// TIA Portal V19 export
FUNCTION "LSW_INTERLOCK" : Void   // FC9, LAD
{ S7_Optimized_Access := 'TRUE' }
// stored: SetENOAutomatically false
   VAR_TEMP   // added for the SCL form of the ladder/FBD networks
      _w1 : Bool;
      _w2 : Bool;
   END_VAR
BEGIN

REGION Network 1: FORWARD LSW
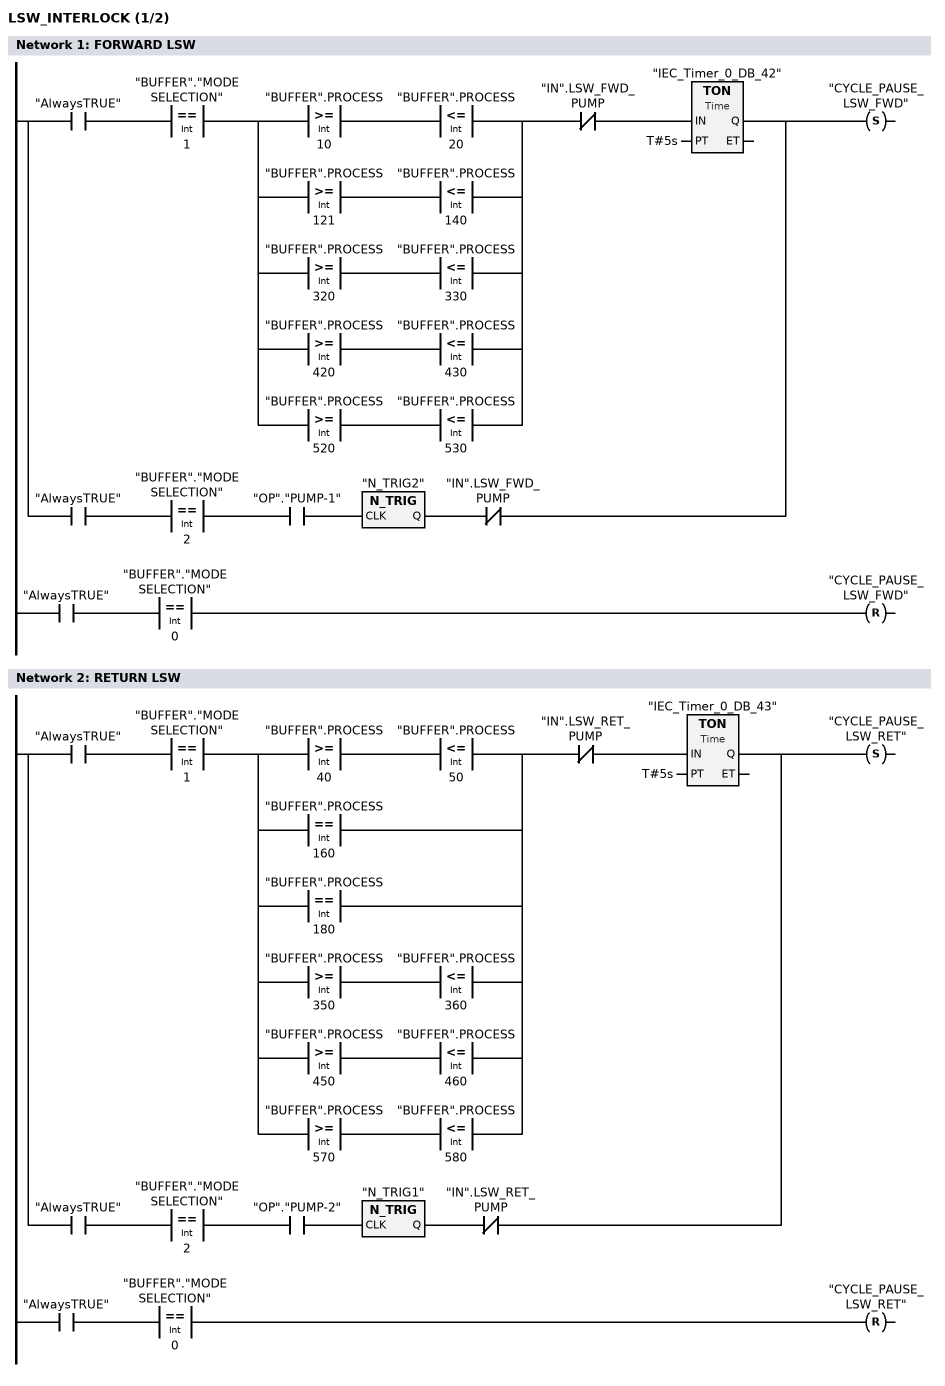
   RUNG wire#powerrail
      Contact( "AlwaysTRUE" )
      { S7_Templates := "SrcType := Int" } EQ_Contact(in1 := "BUFFER"."MODE SELECTION", in2 := 1)
      wire#w1
      { S7_Templates := "SrcType := Int" } GE_Contact(in1 := "BUFFER".PROCESS, in2 := 10)
      { S7_Templates := "SrcType := Int" } LE_Contact(in1 := "BUFFER".PROCESS, in2 := 20)
      wire#w2
      I_Contact( "IN".LSW_FWD_PUMP )
      { S7_Templates := "time_type := Time" } "IEC_Timer_0_DB_42".TON(pt := T#5s, et =>)
      wire#w3
      S_Coil( "CYCLE_PAUSE_LSW_FWD" )
   END_RUNG
   RUNG wire#w1
      { S7_Templates := "SrcType := Int" } GE_Contact(in1 := "BUFFER".PROCESS, in2 := 121)
      { S7_Templates := "SrcType := Int" } LE_Contact(in1 := "BUFFER".PROCESS, in2 := 140)
   END_RUNG wire#w2
   RUNG wire#w1
      { S7_Templates := "SrcType := Int" } GE_Contact(in1 := "BUFFER".PROCESS, in2 := 320)
      { S7_Templates := "SrcType := Int" } LE_Contact(in1 := "BUFFER".PROCESS, in2 := 330)
   END_RUNG wire#w2
   RUNG wire#w1
      { S7_Templates := "SrcType := Int" } GE_Contact(in1 := "BUFFER".PROCESS, in2 := 420)
      { S7_Templates := "SrcType := Int" } LE_Contact(in1 := "BUFFER".PROCESS, in2 := 430)
   END_RUNG wire#w2
   RUNG wire#w1
      { S7_Templates := "SrcType := Int" } GE_Contact(in1 := "BUFFER".PROCESS, in2 := 520)
      { S7_Templates := "SrcType := Int" } LE_Contact(in1 := "BUFFER".PROCESS, in2 := 530)
   END_RUNG wire#w2
   RUNG wire#powerrail
      Contact( "AlwaysTRUE" )
      { S7_Templates := "SrcType := Int" } EQ_Contact(in1 := "BUFFER"."MODE SELECTION", in2 := 2)
      Contact( "OP"."PUMP-1" )
      N_Trig( "N_TRIG2" )
      I_Contact( "IN".LSW_FWD_PUMP )
   END_RUNG wire#w3
   RUNG wire#powerrail
      Contact( "AlwaysTRUE" )
      { S7_Templates := "SrcType := Int" } EQ_Contact(in1 := "BUFFER"."MODE SELECTION", in2 := 0)
      R_Coil( "CYCLE_PAUSE_LSW_FWD" )
   END_RUNG
   // the same network as SCL:
   "IEC_Timer_0_DB_42".TON(IN := "AlwaysTRUE" AND ("BUFFER"."MODE SELECTION" = 1) AND ((("BUFFER".PROCESS >= 10) AND ("BUFFER".PROCESS <= 20)) OR (("BUFFER".PROCESS >= 121) AND ("BUFFER".PROCESS <= 140)) OR (("BUFFER".PROCESS >= 320) AND ("BUFFER".PROCESS <= 330)) OR (("BUFFER".PROCESS >= 420) AND ("BUFFER".PROCESS <= 430)) OR (("BUFFER".PROCESS >= 520) AND ("BUFFER".PROCESS <= 530))) AND NOT "IN".LSW_FWD_PUMP,
                           PT := T#5s);
   #_w1 := "AlwaysTRUE" AND ("BUFFER"."MODE SELECTION" = 2) AND "OP"."PUMP-1";
   #_w2 := NOT #_w1 AND "N_TRIG2";   // falling edge
   "N_TRIG2" := #_w1;
   IF "IEC_Timer_0_DB_42".Q OR (#_w2 AND NOT "IN".LSW_FWD_PUMP) THEN "CYCLE_PAUSE_LSW_FWD" := TRUE; END_IF;
   IF "AlwaysTRUE" AND ("BUFFER"."MODE SELECTION" = 0) THEN "CYCLE_PAUSE_LSW_FWD" := FALSE; END_IF;
END_REGION

REGION Network 2: RETURN LSW
   RUNG wire#powerrail
      Contact( "AlwaysTRUE" )
      { S7_Templates := "SrcType := Int" } EQ_Contact(in1 := "BUFFER"."MODE SELECTION", in2 := 1)
      wire#w1
      { S7_Templates := "SrcType := Int" } GE_Contact(in1 := "BUFFER".PROCESS, in2 := 40)
      { S7_Templates := "SrcType := Int" } LE_Contact(in1 := "BUFFER".PROCESS, in2 := 50)
      wire#w2
      I_Contact( "IN".LSW_RET_PUMP )
      { S7_Templates := "time_type := Time" } "IEC_Timer_0_DB_43".TON(pt := T#5s, et =>)
      wire#w3
      S_Coil( "CYCLE_PAUSE_LSW_RET" )
   END_RUNG
   RUNG wire#w1
      { S7_Templates := "SrcType := Int" } EQ_Contact(in1 := "BUFFER".PROCESS, in2 := 160)
   END_RUNG wire#w2
   RUNG wire#w1
      { S7_Templates := "SrcType := Int" } EQ_Contact(in1 := "BUFFER".PROCESS, in2 := 180)
   END_RUNG wire#w2
   RUNG wire#w1
      { S7_Templates := "SrcType := Int" } GE_Contact(in1 := "BUFFER".PROCESS, in2 := 350)
      { S7_Templates := "SrcType := Int" } LE_Contact(in1 := "BUFFER".PROCESS, in2 := 360)
   END_RUNG wire#w2
   RUNG wire#w1
      { S7_Templates := "SrcType := Int" } GE_Contact(in1 := "BUFFER".PROCESS, in2 := 450)
      { S7_Templates := "SrcType := Int" } LE_Contact(in1 := "BUFFER".PROCESS, in2 := 460)
   END_RUNG wire#w2
   RUNG wire#w1
      { S7_Templates := "SrcType := Int" } GE_Contact(in1 := "BUFFER".PROCESS, in2 := 570)
      { S7_Templates := "SrcType := Int" } LE_Contact(in1 := "BUFFER".PROCESS, in2 := 580)
   END_RUNG wire#w2
   RUNG wire#powerrail
      Contact( "AlwaysTRUE" )
      { S7_Templates := "SrcType := Int" } EQ_Contact(in1 := "BUFFER"."MODE SELECTION", in2 := 2)
      Contact( "OP"."PUMP-2" )
      N_Trig( "N_TRIG1" )
      I_Contact( "IN".LSW_RET_PUMP )
   END_RUNG wire#w3
   RUNG wire#powerrail
      Contact( "AlwaysTRUE" )
      { S7_Templates := "SrcType := Int" } EQ_Contact(in1 := "BUFFER"."MODE SELECTION", in2 := 0)
      R_Coil( "CYCLE_PAUSE_LSW_RET" )
   END_RUNG
   // the same network as SCL:
   "IEC_Timer_0_DB_43".TON(IN := "AlwaysTRUE" AND ("BUFFER"."MODE SELECTION" = 1) AND ((("BUFFER".PROCESS >= 40) AND ("BUFFER".PROCESS <= 50)) OR ("BUFFER".PROCESS = 160) OR ("BUFFER".PROCESS = 180) OR (("BUFFER".PROCESS >= 350) AND ("BUFFER".PROCESS <= 360)) OR (("BUFFER".PROCESS >= 450) AND ("BUFFER".PROCESS <= 460)) OR (("BUFFER".PROCESS >= 570) AND ("BUFFER".PROCESS <= 580))) AND NOT "IN".LSW_RET_PUMP,
                           PT := T#5s);
   #_w1 := "AlwaysTRUE" AND ("BUFFER"."MODE SELECTION" = 2) AND "OP"."PUMP-2";
   #_w2 := NOT #_w1 AND "N_TRIG1";   // falling edge
   "N_TRIG1" := #_w1;
   IF "IEC_Timer_0_DB_43".Q OR (#_w2 AND NOT "IN".LSW_RET_PUMP) THEN "CYCLE_PAUSE_LSW_RET" := TRUE; END_IF;
   IF "AlwaysTRUE" AND ("BUFFER"."MODE SELECTION" = 0) THEN "CYCLE_PAUSE_LSW_RET" := FALSE; END_IF;
END_REGION

REGION Network 3: cycle pause
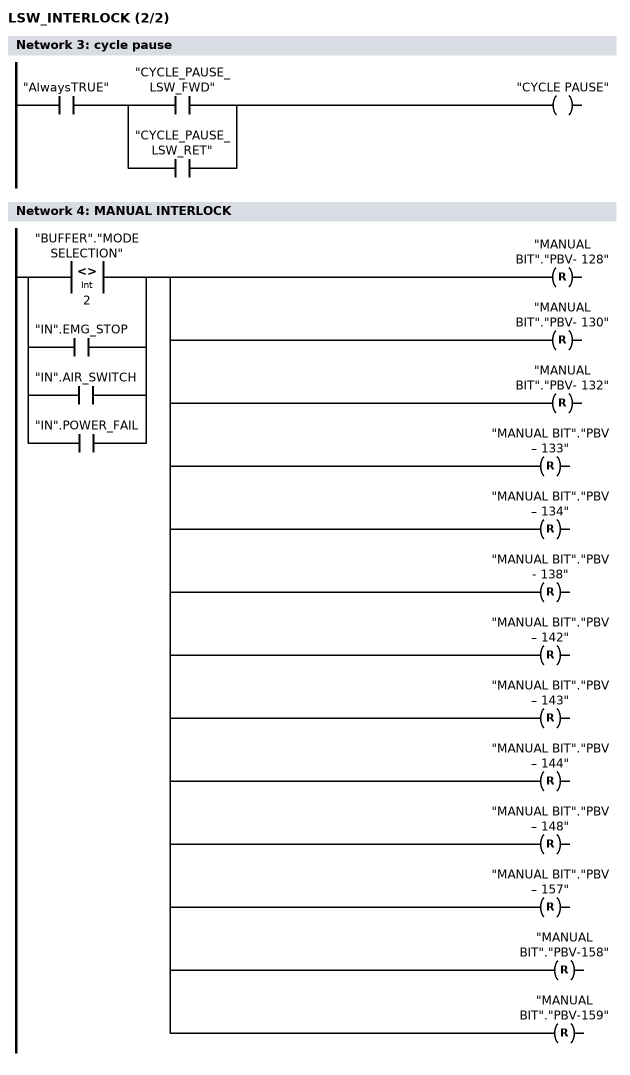
   RUNG wire#powerrail
      Contact( "AlwaysTRUE" )
      wire#w1
      Contact( "CYCLE_PAUSE_LSW_FWD" )
      wire#w2
      Coil( "CYCLE PAUSE" )
   END_RUNG
   RUNG wire#w1
      Contact( "CYCLE_PAUSE_LSW_RET" )
   END_RUNG wire#w2
   // the same network as SCL:
   "CYCLE PAUSE" := "AlwaysTRUE" AND ("CYCLE_PAUSE_LSW_FWD" OR "CYCLE_PAUSE_LSW_RET");
END_REGION

REGION Network 4: MANUAL INTERLOCK
   RUNG wire#powerrail
      { S7_Templates := "SrcType := Int" } NE_Contact(in1 := "BUFFER"."MODE SELECTION", in2 := 2)
      wire#w1
      R_Coil( "MANUAL BIT"."PBV- 128" )
   END_RUNG
   RUNG wire#powerrail
      Contact( "IN".EMG_STOP )
   END_RUNG wire#w1
   RUNG wire#powerrail
      Contact( "IN".AIR_SWITCH )
   END_RUNG wire#w1
   RUNG wire#powerrail
      Contact( "IN".POWER_FAIL )
   END_RUNG wire#w1
   RUNG wire#w1
      R_Coil( "MANUAL BIT"."PBV- 130" )
   END_RUNG
   RUNG wire#w1
      R_Coil( "MANUAL BIT"."PBV- 132" )
   END_RUNG
   RUNG wire#w1
      R_Coil( "MANUAL BIT"."PBV – 133" )
   END_RUNG
   RUNG wire#w1
      R_Coil( "MANUAL BIT"."PBV – 134" )
   END_RUNG
   RUNG wire#w1
      R_Coil( "MANUAL BIT"."PBV - 138" )
   END_RUNG
   RUNG wire#w1
      R_Coil( "MANUAL BIT"."PBV – 142" )
   END_RUNG
   RUNG wire#w1
      R_Coil( "MANUAL BIT"."PBV – 143" )
   END_RUNG
   RUNG wire#w1
      R_Coil( "MANUAL BIT"."PBV – 144" )
   END_RUNG
   RUNG wire#w1
      R_Coil( "MANUAL BIT"."PBV – 148" )
   END_RUNG
   RUNG wire#w1
      R_Coil( "MANUAL BIT"."PBV – 157" )
   END_RUNG
   RUNG wire#w1
      R_Coil( "MANUAL BIT"."PBV-158" )
   END_RUNG
   RUNG wire#w1
      R_Coil( "MANUAL BIT"."PBV-159" )
   END_RUNG
   // the same network as SCL:
   IF ("BUFFER"."MODE SELECTION" <> 2) OR "IN".EMG_STOP OR "IN".AIR_SWITCH OR "IN".POWER_FAIL THEN
       "MANUAL BIT"."PBV- 128" := FALSE;
       "MANUAL BIT"."PBV- 130" := FALSE;
       "MANUAL BIT"."PBV- 132" := FALSE;
       "MANUAL BIT"."PBV – 133" := FALSE;
       "MANUAL BIT"."PBV – 134" := FALSE;
       "MANUAL BIT"."PBV - 138" := FALSE;
       "MANUAL BIT"."PBV – 142" := FALSE;
       "MANUAL BIT"."PBV – 143" := FALSE;
       "MANUAL BIT"."PBV – 144" := FALSE;
       "MANUAL BIT"."PBV – 148" := FALSE;
       "MANUAL BIT"."PBV – 157" := FALSE;
       "MANUAL BIT"."PBV-158" := FALSE;
       "MANUAL BIT"."PBV-159" := FALSE;
   END_IF;
END_REGION
END_FUNCTION
